// TIA Portal project "Box_Count" (V18)

(* hardware
DEVICE "S7-1200 station_1"  S7-1200 Station
   slot 0: "Rack_0"  S7-1200 Rack  Rack  V1.0
   slot 1: "PLC_1"  CPU 1214C DC/DC/DC  6ES7 214-1AG40-0XB0  V4.6
*)

// ===== PLC "PLC_1"  CPU 1214C DC/DC/DC =====

VAR_GLOBAL   // PLC tag table "Default tag table"
   "Start_Button" AT %M0.0 : Bool;
   "Convoyer_Motor" AT %Q0.0 : Bool;
   "Stop_Button" AT %I0.1 : Bool;
   "Proxi_Sensor" AT %M0.2 : Bool;
   "Rising Edge Detection Bit" AT %M0.3 : Bool;
   "Current Value" AT %MW10 : Word;
   "Counter Done Bit" AT %M0.4 : Bool;
END_VAR

// folder: System blocks/Program resources

DATA_BLOCK "IEC_Counter_0_DB"   // DB1
{ S7_Optimized_Access := 'TRUE' }
AUTHOR : Simatic
FAMILY : IEC
NAME : CNTR
VERSION : 1.0
// stored: InstanceOfName IEC_COUNTER
"IEC_COUNTER"
BEGIN
END_DATA_BLOCK

// folder: (top level)

ORGANIZATION_BLOCK "Main"   // OB1, LAD, ProgramCycle
TITLE = "Main Program Sweep (Cycle)"
{ S7_Optimized_Access := 'TRUE' }
VERSION : 0.1
   VAR_INPUT
      Initial_Call : Bool;   // Initial call of this OB
      Remanence : Bool;   // =True, if remanent data are available
   END_VAR
   VAR_TEMP   // added for the SCL form of the ladder/FBD networks
      _w1 : Bool;
      _w2 : Bool;
   END_VAR
BEGIN

REGION Network 1
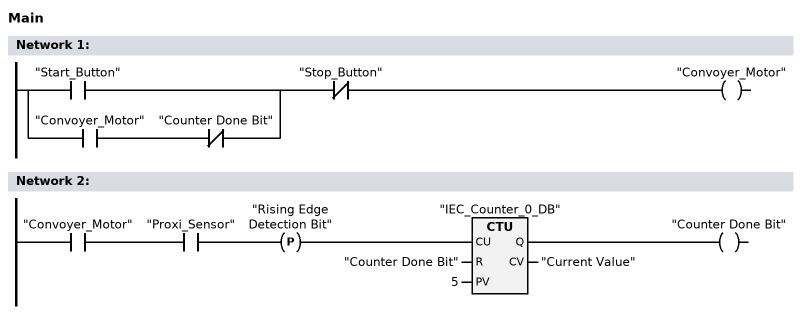
   RUNG wire#powerrail
      Contact( "Start_Button" )
      wire#w1
      I_Contact( "Stop_Button" )
      Coil( "Convoyer_Motor" )
   END_RUNG
   RUNG wire#powerrail
      Contact( "Convoyer_Motor" )
      I_Contact( "Counter Done Bit" )
   END_RUNG wire#w1
   // the same network as SCL:
   "Convoyer_Motor" := ("Start_Button" OR ("Convoyer_Motor" AND NOT "Counter Done Bit")) AND NOT "Stop_Button";
END_REGION

REGION Network 2
   #_w1 := "Convoyer_Motor" AND "Proxi_Sensor";
   #_w2 := #_w1 AND NOT "Rising Edge Detection Bit";   // rising edge
   "Rising Edge Detection Bit" := #_w1;
   "IEC_Counter_0_DB".CTU(CU := #_w2, R := "Counter Done Bit", PV := 5, CV => "Current Value");
   "Counter Done Bit" := "IEC_Counter_0_DB".Q;
END_REGION
END_ORGANIZATION_BLOCK